// TIA Portal V20 export
DATA_BLOCK "SP509"   // DB325
// stored: MemoryReserve 100
   VAR
      "QR MARKING SHUTTER CONTROL INPUT A" : Bool;
      "QR MARKING SHUTTER CONTROL INPUT B" : Bool;
      SPARE : Bool;
      SPARE_1 : Bool;
      SPARE_2 : Bool;
      SPARE_3 : Bool;
      SPARE_4 : Bool;
      SPARE_5 : Bool;
   END_VAR
BEGIN
END_DATA_BLOCK
